FUNCTION_BLOCK Control_Pannel
VAR_INPUT
	OperStart		: BOOL;
	OperReset		: BOOL;
	OperStop		: BOOL;
	AutoManSwitch	: BOOL;
	Interlock		: BOOL;

	
END_VAR
VAR_OUTPUT
	
	LightStart		: BOOL;
	LightStop		: BOOL;
	LightReset		: BOOL;

END_VAR
VAR
	StatusAutoMan	: BOOL;
	Idling			: BOOL;
	Executing		: BOOL;
	Stopping		: BOOL;
	Clock_Bit_Flashing	: BOOL;
	Clock_ON: ton;
	Clock_OFF: ton;

END_VAR
VAR // added by the converter: edge detectors and wires of the graphical bodies
    _w1 : BOOL;
END_VAR

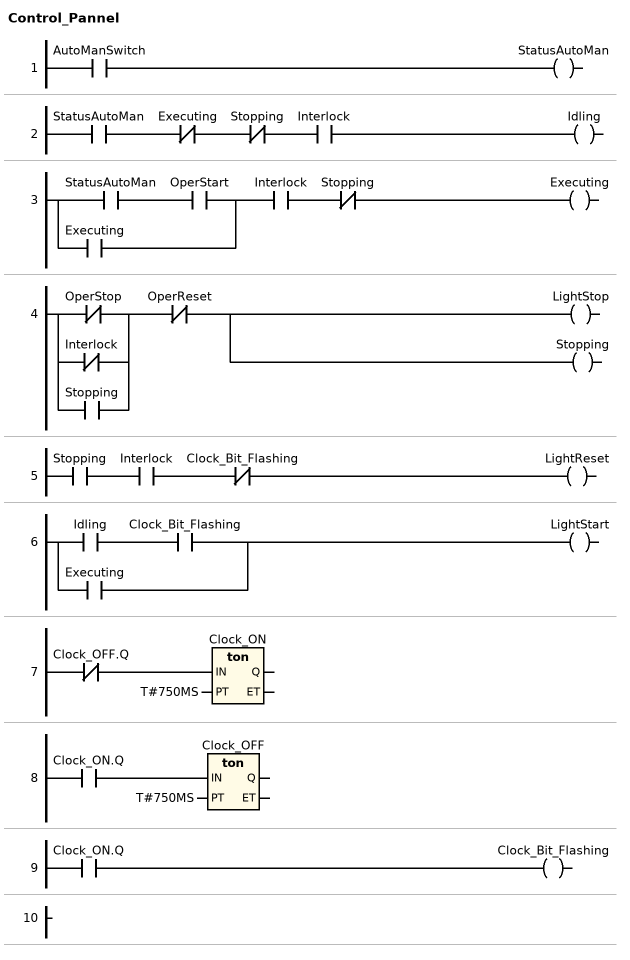
// NETWORK 1
StatusAutoMan := AutoManSwitch;

// NETWORK 2
Idling := StatusAutoMan AND NOT Executing AND NOT Stopping AND Interlock;

// NETWORK 3
Executing := (StatusAutoMan AND OperStart OR Executing) AND Interlock AND NOT Stopping;

// NETWORK 4
_w1 := (NOT OperStop OR NOT Interlock OR Stopping) AND NOT OperReset;
LightStop := _w1;
Stopping := _w1;

// NETWORK 5
LightReset := Stopping AND Interlock AND NOT Clock_Bit_Flashing;

// NETWORK 6
LightStart := Idling AND Clock_Bit_Flashing OR Executing;

// NETWORK 7
Clock_ON(IN := NOT Clock_OFF.Q, PT := T#750MS); // ton

// NETWORK 8
Clock_OFF(IN := Clock_ON.Q, PT := T#750MS); // ton

// NETWORK 9
Clock_Bit_Flashing := Clock_ON.Q;

// NETWORK 10

END_FUNCTION_BLOCK

(* stored: Version 1.1.0.1, ProductVersion 3.1.4024.12
   POU Control_Pannel: Id {174463ef-c7fd-4edf-b1ea-01cdca75283b}, SpecialFunc None *)
